FUNCTION F_ReadAndClear : BOOL {warning 'Depreciated - use F_ReadFlag'} 
VAR_IN_OUT
	Flag : BOOL;
END_VAR

F_ReadAndClear := Flag;
Flag           := FALSE;

END_FUNCTION

(* stored: Version 1.1.0.1, ProductVersion 3.1.4024.12
   POU F_ReadAndClear: Id {463f69b5-0d65-483a-9f34-d8ace50c5d79}, SpecialFunc None *)
